(* PLC project Unnamed, Unknown Unnamed 1 *)
(* stored: creationDateTime 2026-07-04T15:38:14, modificationDateTime 2026-07-04T15:38:14 *)

TYPE ERRORCODES_ENUM : (NO_ERRORS, WRITE_FAIL, VERIFY_FAIL, NO_NODES_FOUND, DUP_SERIAL);
END_TYPE

FUNCTION_BLOCK D64PROGRAMMER_FB
  VAR_INPUT
    I_Execute : BOOL;  (* Rising edge starts the whole sequence *)
    I_TargetCurrent : UDINT;  (* Target current in mA *)
    I_ResponseDelay : UDINT;  (* Response delay in ms *)
  END_VAR
  VAR_OUTPUT
    O_Busy : BOOL;  (* TRUE while scanning/programming *)
    O_Done : BOOL;  (* TRUE when everything passes *)
    O_Error : BOOL;  (* TRUE if any step fails *)
    O_ErrorCode : INT;  (* 0=No Errors, 1=Write Fail, 2=Verify Fail, 3=No Nodes Found, 4=Dup Serial *)
    O_TotalNodes : INT;  (* Total number of D64s found and programmed *)
    O_FailedNodeAddr : INT;  (* The specific Modbus address that caused an error *)
  END_VAR

            /* ================================================================
 * D64 Modbus RTU - Unified Sequencer (Scan -> Program -> Verify)
 * ================================================================ */

#include <Arduino.h> 

static uint8_t  state = 0;
static uint32_t state_timer = 0;
static uint8_t  request[16];
static uint8_t  response[64];
static uint8_t  rx_idx = 0;

static uint8_t  current_addr = 100;
static uint8_t  found_idx = 0;
static uint8_t  node_idx = 0; // Used to iterate through found nodes
static bool     seq_latched = false;

// Arrays to hold discovered nodes during the cycle
static uint8_t valid_nodes[50];
static char    internal_serials[50][33]; 

// -- Hardcoded Verification Targets --
const uint16_t TARGET_MODE = 1;


uint16_t calcCRC(uint8_t *buf, uint16_t len) {
    uint16_t crc = 0xFFFF;
    for (uint16_t pos = 0; pos < len; pos++) {
        crc ^= (uint16_t)buf[pos];
        for (uint8_t i = 8; i != 0; i--) {
            if ((crc & 0x0001) != 0) crc = (crc >> 1) ^ 0xA001;
            else crc >>= 1;
        }
    }
    return crc;
}

void setup() {
    Serial.begin(115200);
    Serial2.begin(19200, SERIAL_8E1, 16, 17);
    
    O_Busy = false;
    O_Done = false;
    O_Error = false;
    O_ErrorCode = 0;
    O_TotalNodes = 0;
    O_FailedNodeAddr = 0;
    seq_latched = false;
    state = 0; 
}

void loop() {
    // 1. Edge Detection & Initialization
    if (I_Execute && !seq_latched) {
        seq_latched = true;
        O_Busy = true;
        O_Done = false;
        O_Error = false;
        O_ErrorCode = 0;
        O_TotalNodes = 0;
        O_FailedNodeAddr = 0;
        
        current_addr = 100; 
        found_idx = 0;      
        state = 1; // Start Scan Phase
    }
    
    if (!I_Execute) seq_latched = false;

    switch (state) {
        case 0: break; // IDLE

        // ==========================================
        // PHASE 1: DISCOVERY & DUPLICATE CHECK
        // ==========================================
        case 1: { // REQUEST SERIAL
            request[0] = current_addr;
            request[1] = 0x03; 
            request[2] = 0x00; request[3] = 0x20; 
            request[4] = 0x00; request[5] = 0x10; 
            
            uint16_t crc = calcCRC(request, 6);
            request[6] = crc & 0xFF; request[7] = crc >> 8;

            while(Serial2.available()) Serial2.read(); 
            Serial2.write(request, 8);
            
            rx_idx = 0;             
            state_timer = millis(); 
            state = 2;              
            break;
        } 

        case 2: { // WAIT FOR SERIAL
            while (Serial2.available() && rx_idx < 64) response[rx_idx++] = Serial2.read();

            if (rx_idx >= 5 && response[1] == 0x03) {
                uint8_t expected_len = 5 + response[2]; 
                if (rx_idx >= expected_len) {
                    
                    uint8_t byteCount = response[2];
                    if (byteCount > 32) byteCount = 32; 
                    
                    for (uint8_t i = 0; i < byteCount; i++) {
                        internal_serials[found_idx][i] = response[3 + i];
                    }
                    internal_serials[found_idx][byteCount] = '\0'; 
                    valid_nodes[found_idx] = current_addr;
                    found_idx++;
                    
                    state_timer = millis(); 
                    state = 3; 
                    break; 
                }
            }
            if (millis() - state_timer > 150) state = 3; // Timeout, node missing, skip
            break;
        } 

        case 3: { // NEXT ADDRESS / VALIDATE SCAN
            current_addr++;
            if (current_addr > 199 || found_idx >= 50) {
                
                if (found_idx == 0) {
                    O_ErrorCode = 3; // Error: No Nodes Found
                    state = 99;
                    break;
                }

                // Check Duplicates
                bool dup = false;
                if (found_idx > 1) {
                    for (int i = 0; i < found_idx - 1; i++) {
                        for (int j = i + 1; j < found_idx; j++) {
                            if (strcmp(internal_serials[i], internal_serials[j]) == 0) dup = true;
                        }
                    }
                }
                
                if (dup) {
                    O_ErrorCode = 4; // Error: Duplicate Serials
                    state = 99;
                } else {
                    O_TotalNodes = found_idx;
                    node_idx = 0;
                    state = 10; // Move to Programming Phase
                }
            } else {
                state = 1; // Ping next addr
            }
            break;
        }

        // ==========================================
        // PHASE 2: PROGRAMMING
        // ==========================================
        case 10: { // WRITE MODE (32101 = TARGET_MODE)
            request[0] = valid_nodes[node_idx];
            request[1] = 0x10; 
            request[2] = 0x7D; request[3] = 0x65; 
            request[4] = 0x00; request[5] = 0x01; 
            request[6] = 0x02; 
            request[7] = (TARGET_MODE >> 8) & 0xFF; 
            request[8] = TARGET_MODE & 0xFF; 
            
            uint16_t crc = calcCRC(request, 9);
            request[9] = crc & 0xFF; request[10] = crc >> 8;

            while(Serial2.available()) Serial2.read(); 
            Serial2.write(request, 11);
            
            rx_idx = 0;             
            state_timer = millis(); 
            state = 11;              
            break;
        }

        case 11: { // WAIT WRITE MODE
            if (Serial2.available() >= 8) {
                state = 12;
            } else if (millis() - state_timer > 600) {
                O_ErrorCode = 1; // Write Timeout
                O_FailedNodeAddr = valid_nodes[node_idx];
                state = 99;
            }
            break;
        }

        case 12: { // WRITE CURRENT (32107 = I_TargetCurrent)
            request[0] = valid_nodes[node_idx];
            request[1] = 0x10; 
            request[2] = 0x7D; request[3] = 0x6B; 
            request[4] = 0x00; request[5] = 0x02; 
            request[6] = 0x04; 
            request[7] = (I_TargetCurrent >> 24) & 0xFF; request[8] = (I_TargetCurrent >> 16) & 0xFF; 
            request[9] = (I_TargetCurrent >> 8) & 0xFF;  request[10] = I_TargetCurrent & 0xFF; 
            
            uint16_t crc = calcCRC(request, 11);
            request[11] = crc & 0xFF; request[12] = crc >> 8;

            while(Serial2.available()) Serial2.read(); 
            Serial2.write(request, 13);
            
            state_timer = millis(); 
            state = 13;              
            break;
        }

        case 13: { // WAIT WRITE CURRENT
            if (Serial2.available() >= 8) {
                state = 14; // Go to WRITE DELAY
            } else if (millis() - state_timer > 600) {
                O_ErrorCode = 1; 
                O_FailedNodeAddr = valid_nodes[node_idx];
                state = 99;
            }
            break;
        }

        case 14: { // WRITE DELAY (32112 = I_ResponseDelay)
            request[0] = valid_nodes[node_idx];
            request[1] = 0x10; 
            request[2] = 0x7D; request[3] = 0x70; 
            request[4] = 0x00; request[5] = 0x02; 
            request[6] = 0x04; 
            request[7] = (I_ResponseDelay >> 24) & 0xFF; request[8] = (I_ResponseDelay >> 16) & 0xFF; 
            request[9] = (I_ResponseDelay >> 8) & 0xFF;  request[10] = I_ResponseDelay & 0xFF; 
            
            uint16_t crc = calcCRC(request, 11);
            request[11] = crc & 0xFF; request[12] = crc >> 8;

            while(Serial2.available()) Serial2.read(); 
            Serial2.write(request, 13);
            
            state_timer = millis(); 
            state = 15;              
            break;
        }

        case 15: { // WAIT WRITE DELAY
            if (Serial2.available() >= 8) {
                node_idx++;
                if (node_idx >= found_idx) {
                    node_idx = 0;
                    state = 20; // Move to Verification Phase
                } else {
                    state = 10; // Program next node
                }
            } else if (millis() - state_timer > 600) {
                O_ErrorCode = 1; 
                O_FailedNodeAddr = valid_nodes[node_idx];
                state = 99;
            }
            break;
        }

        // ==========================================
        // PHASE 3: VERIFICATION
        // ==========================================
        case 20: { // READ MODE
            request[0] = valid_nodes[node_idx];
            request[1] = 0x03; 
            request[2] = 0x7D; request[3] = 0x65; 
            request[4] = 0x00; request[5] = 0x01; 
            
            uint16_t crc = calcCRC(request, 6);
            request[6] = crc & 0xFF; request[7] = crc >> 8;

            while(Serial2.available()) Serial2.read(); 
            Serial2.write(request, 8);
            
            rx_idx = 0;             
            state_timer = millis(); 
            state = 21;              
            break;
        }

        case 21: { // VERIFY MODE
            while (Serial2.available() && rx_idx < 64) response[rx_idx++] = Serial2.read();

            if (rx_idx >= 5 && response[1] == 0x03) {
                uint8_t expected = 5 + response[2]; 
                if (rx_idx >= expected) {
                    uint16_t read_mode = (response[3] << 8) | response[4];
                    if (read_mode != TARGET_MODE) {
                        O_ErrorCode = 2; // Verify Failed
                        O_FailedNodeAddr = valid_nodes[node_idx];
                        state = 99;
                    } else {
                        state = 22;
                    }
                    break;
                }
            }
            if (millis() - state_timer > 600) { O_ErrorCode = 1; O_FailedNodeAddr = valid_nodes[node_idx]; state = 99; }
            break;
        }

        case 22: { // READ CURRENT
            request[0] = valid_nodes[node_idx];
            request[1] = 0x03; 
            request[2] = 0x7D; request[3] = 0x6B; 
            request[4] = 0x00; request[5] = 0x02; 
            
            uint16_t crc = calcCRC(request, 6);
            request[6] = crc & 0xFF; request[7] = crc >> 8;

            while(Serial2.available()) Serial2.read(); 
            Serial2.write(request, 8);
            
            rx_idx = 0;             
            state_timer = millis(); 
            state = 23;              
            break;
        }

        case 23: { // VERIFY CURRENT
            while (Serial2.available() && rx_idx < 64) response[rx_idx++] = Serial2.read();

            if (rx_idx >= 5 && response[1] == 0x03) {
                uint8_t expected = 5 + response[2]; 
                if (rx_idx >= expected) {
                    uint32_t read_current = (response[3] << 24) | (response[4] << 16) | (response[5] << 8) | response[6];
                    if (read_current != I_TargetCurrent) {
                        O_ErrorCode = 2; // Verify Failed
                        O_FailedNodeAddr = valid_nodes[node_idx];
                        state = 99;
                    } else {
                        state = 24; // VERIFY DELAY
                    }
                    break;
                }
            }
            if (millis() - state_timer > 600) { O_ErrorCode = 1; O_FailedNodeAddr = valid_nodes[node_idx]; state = 99; }
            break;
        }

        case 24: { // READ DELAY
            request[0] = valid_nodes[node_idx];
            request[1] = 0x03; 
            request[2] = 0x7D; request[3] = 0x70; 
            request[4] = 0x00; request[5] = 0x02; 
            
            uint16_t crc = calcCRC(request, 6);
            request[6] = crc & 0xFF; request[7] = crc >> 8;

            while(Serial2.available()) Serial2.read(); 
            Serial2.write(request, 8);
            
            rx_idx = 0;             
            state_timer = millis(); 
            state = 25;              
            break;
        }

        case 25: { // VERIFY DELAY
            while (Serial2.available() && rx_idx < 64) response[rx_idx++] = Serial2.read();

            if (rx_idx >= 5 && response[1] == 0x03) {
                uint8_t expected = 5 + response[2]; 
                if (rx_idx >= expected) {
                    uint32_t read_delay = (response[3] << 24) | (response[4] << 16) | (response[5] << 8) | response[6];
                    if (read_delay != I_ResponseDelay) {
                        O_ErrorCode = 2; // Verify Failed
                        O_FailedNodeAddr = valid_nodes[node_idx];
                        state = 99;
                    } else {
                        node_idx++;
                        if (node_idx >= found_idx) {
                            O_Done = true; // ENTIRE PROCESS COMPLETE!
                            state = 99;
                        } else {
                            state = 20; // Verify next node
                        }
                    }
                    break;
                }
            }
            if (millis() - state_timer > 600) { O_ErrorCode = 1; O_FailedNodeAddr = valid_nodes[node_idx]; state = 99; }
            break;
        }

        // ==========================================
        // FINISH / ABORT
        // ==========================================
        case 99: { 
            O_Busy = false;
            if (O_ErrorCode > 0) O_Error = true;
            
            // Wait for user to release the I_Execute button
            if (!I_Execute) {
                seq_latched = false;
                state = 0;
            }
            break;
        } 
    }
}
          
END_FUNCTION_BLOCK

FUNCTION_BLOCK ReadInputs_FB
  VAR_OUTPUT
    O_BtnStart : BOOL;  (* Debounced output for the Start sequence *)
  END_VAR

            /* ================================================================
 * C/C++ FUNCTION BLOCK : Hardware INIT & Debounce
 * ================================================================ */
#include <stdio.h>
#include <stdint.h>
#include <stdbool.h>
#include <Arduino.h>

// Called once when the block is initialized
void setup()
{
    // --- Configure Input Pins ---
    // Change '18' to whichever GPIO pin your physical button is wired to
    pinMode(18, INPUT_PULLDOWN);   // BtnStart 

    // --- Configure LED Output Pins ---
    // Change these to match your LED GPIO pins. 
    // Initializing them here prevents them from flashing randomly on boot.
    pinMode(19, OUTPUT);           // Busy LED 
    pinMode(21, OUTPUT);           // Done LED
    pinMode(22, OUTPUT);           // Error LED

    digitalWrite(19, LOW);
    digitalWrite(21, LOW);
    digitalWrite(22, LOW);

    printf("BoardINIT: Pins configured with software debounce\n");
}

// Called at every PLC scan cycle
void loop()
{
    static unsigned long lastDebounceTime = 0;
    static bool          lastButtonState  = false;
    static bool          buttonState      = false;

    // Read the raw physical pin
    bool raw = digitalRead(18);

    // Reset the debounce timer if the state changed (noise or actual press)
    if (raw != lastButtonState) {
        lastDebounceTime = millis();
    }

    // If the state has been stable longer than 50ms, lock it in
    if ((millis() - lastDebounceTime) > 50) {   
        if (raw != buttonState) {
            buttonState = raw;
        }
    }
    
    lastButtonState = raw;

    // Output the clean, debounced state to the OpenPLC engine
    O_BtnStart = buttonState;
}
          
END_FUNCTION_BLOCK

PROGRAM main
  VAR
    LedBusy AT %QX0.0 : BOOL;
    LedDone AT %QX0.1 : BOOL;
    LedError AT %QX0.2 : BOOL;
  END_VAR
  VAR
    ReadInputs : READINPUTS_FB;
    Start : BOOL;
    Programmer : D64PROGRAMMER_FB;
    Error : INT;
    NodesProgrammed : INT;
    FailedNode : INT;
    SetTargetCurrent : UDINT := 30;
    SetResponseDelay : UDINT := 0;
    ErrorCodes : ERRORCODES_ENUM;
  END_VAR

            // ==============================================================================
// 1. HARDWARE I/O READ
// ==============================================================================
// Call the block to run the C++ debounce logic
ReadInputs(O_BtnStart => Start);

// ==============================================================================
// 2. D64 MASTER PROGRAMMER LOGIC
// ==============================================================================
// Pass the debounced physical button directly into the sequencer's Execute pin
Programmer(I_Execute := Start,
           I_TargetCurrent := SetTargetCurrent,
           I_ResponseDelay := SetResponseDelay,
           O_Busy => LedBusy,
           O_Done => LedDone,
           O_Error => LedError,
           O_ErrorCode => Error,
           O_TotalNodes => NodesProgrammed,
           O_FailedNodeAddr => FailedNode);
          
END_PROGRAM

CONFIGURATION Config0
  RESOURCE Res0 ON PLC
    TASK task0(INTERVAL := T#20ms, PRIORITY := 1);
    PROGRAM instance0 WITH task0 : main;
  END_RESOURCE
END_CONFIGURATION
